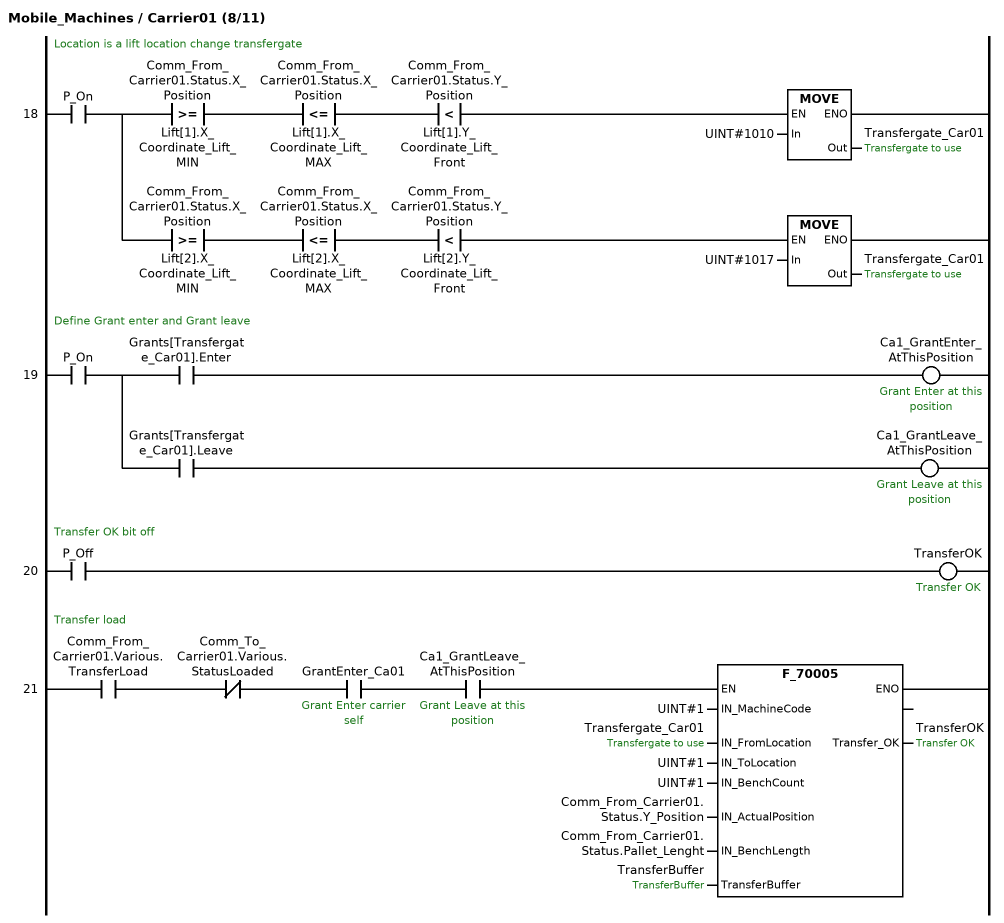
(* [picture p30: Mobile_Machines / Carrier01, rungs 18-21] *)
(* Rung 18: Location is a lift location change transfergate *)
IF P_On AND (Comm_From_Carrier01.Status.X_Position >= Lift[1].X_Coordinate_Lift_MIN) AND (Comm_From_Carrier01.Status.X_Position <= Lift[1].X_Coordinate_Lift_MAX) AND (Comm_From_Carrier01.Status.Y_Position < Lift[1].Y_Coordinate_Lift_Front) THEN
    Transfergate_Car01 := UINT#1010;
END_IF;
IF P_On AND (Comm_From_Carrier01.Status.X_Position >= Lift[2].X_Coordinate_Lift_MIN) AND (Comm_From_Carrier01.Status.X_Position <= Lift[2].X_Coordinate_Lift_MAX) AND (Comm_From_Carrier01.Status.Y_Position < Lift[2].Y_Coordinate_Lift_Front) THEN
    Transfergate_Car01 := UINT#1017;
END_IF;
(* Rung 19: Define Grant enter and Grant leave *)
Ca1_GrantEnter_AtThisPosition := P_On AND Grants[Transfergate_Car01].Enter;
Ca1_GrantLeave_AtThisPosition := P_On AND Grants[Transfergate_Car01].Leave;
(* Rung 20: Transfer OK bit off *)
TransferOK := P_Off;
(* Rung 21: Transfer load *)
IF Comm_From_Carrier01.Various.TransferLoad AND NOT Comm_To_Carrier01.Various.StatusLoaded AND GrantEnter_Ca01 AND Ca1_GrantLeave_AtThisPosition THEN
    F_70005(IN_MachineCode := UINT#1, IN_FromLocation := Transfergate_Car01, IN_ToLocation := UINT#1, IN_BenchCount := UINT#1, IN_ActualPosition := Comm_From_Carrier01.Status.Y_Position, IN_BenchLength := Comm_From_Carrier01.Status.Pallet_Lenght, TransferBuffer := TransferBuffer, Transfer_OK => TransferOK);
END_IF;

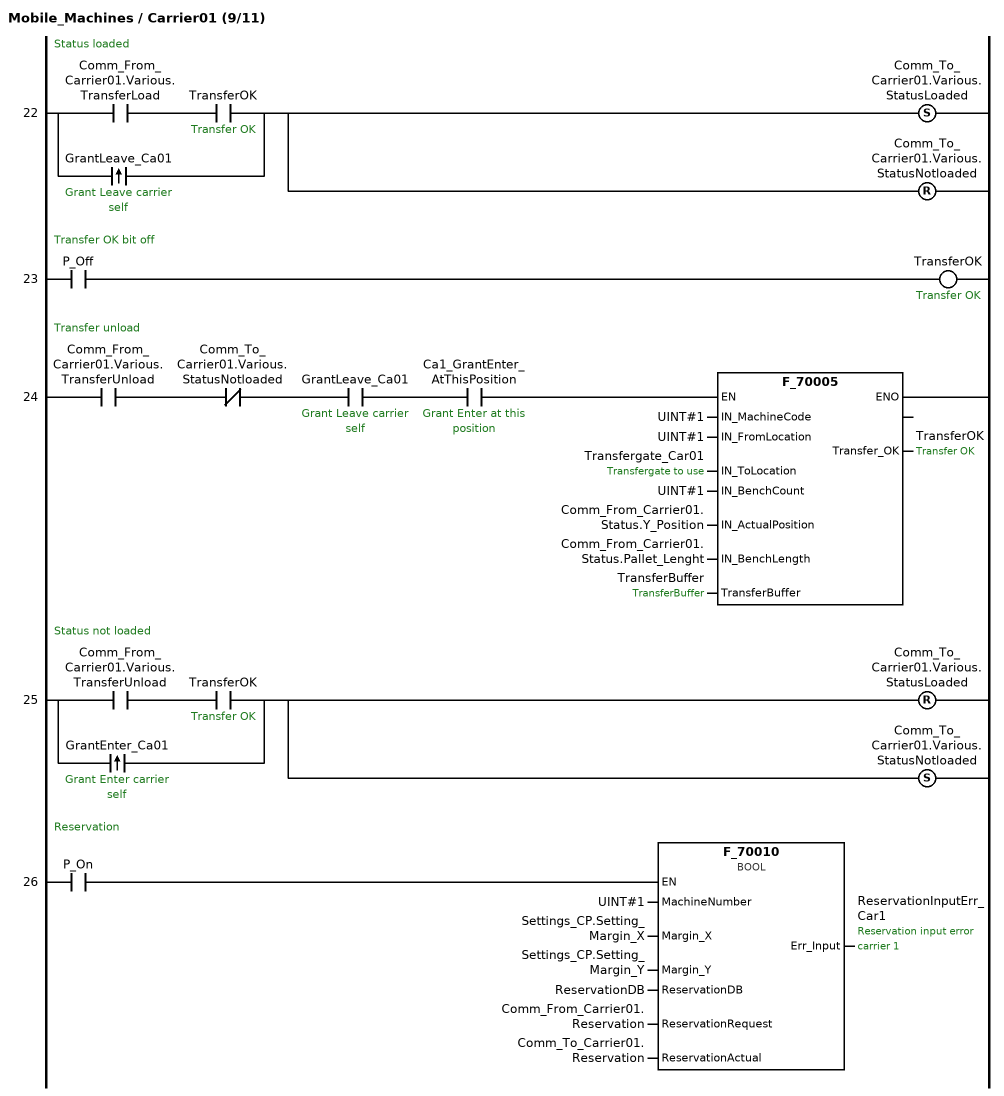
(* Rung 22: Status loaded *)
_e5(CLK := GrantLeave_Ca01);
_p6 := (Comm_From_Carrier01.Various.TransferLoad AND TransferOK) OR _e5.Q;
IF _p6 THEN
    Comm_To_Carrier01.Various.StatusLoaded := TRUE;
    Comm_To_Carrier01.Various.StatusNotloaded := FALSE;
END_IF;
(* Rung 23: Transfer OK bit off *)
TransferOK := P_Off;
(* Rung 24: Transfer unload *)
IF Comm_From_Carrier01.Various.TransferUnload AND NOT Comm_To_Carrier01.Various.StatusNotloaded AND GrantLeave_Ca01 AND Ca1_GrantEnter_AtThisPosition THEN
    F_70005(IN_MachineCode := UINT#1, IN_FromLocation := UINT#1, IN_ToLocation := Transfergate_Car01, IN_BenchCount := UINT#1, IN_ActualPosition := Comm_From_Carrier01.Status.Y_Position, IN_BenchLength := Comm_From_Carrier01.Status.Pallet_Lenght, TransferBuffer := TransferBuffer, Transfer_OK => TransferOK);
END_IF;
(* Rung 25: Status not loaded *)
_e7(CLK := GrantEnter_Ca01);
_p8 := (Comm_From_Carrier01.Various.TransferUnload AND TransferOK) OR _e7.Q;
IF _p8 THEN
    Comm_To_Carrier01.Various.StatusLoaded := FALSE;
    Comm_To_Carrier01.Various.StatusNotloaded := TRUE;
END_IF;
(* Rung 26: Reservation *)
_t9 := FALSE;
IF P_On THEN _t9 := F_70010(MachineNumber := UINT#1, Margin_X := Settings_CP.Setting_Margin_X, Margin_Y := Settings_CP.Setting_Margin_Y, ReservationDB := ReservationDB, ReservationRequest := Comm_From_Carrier01.Reservation, ReservationActual := Comm_To_Carrier01.Reservation, Err_Input => ReservationInputErr_Car1); END_IF;

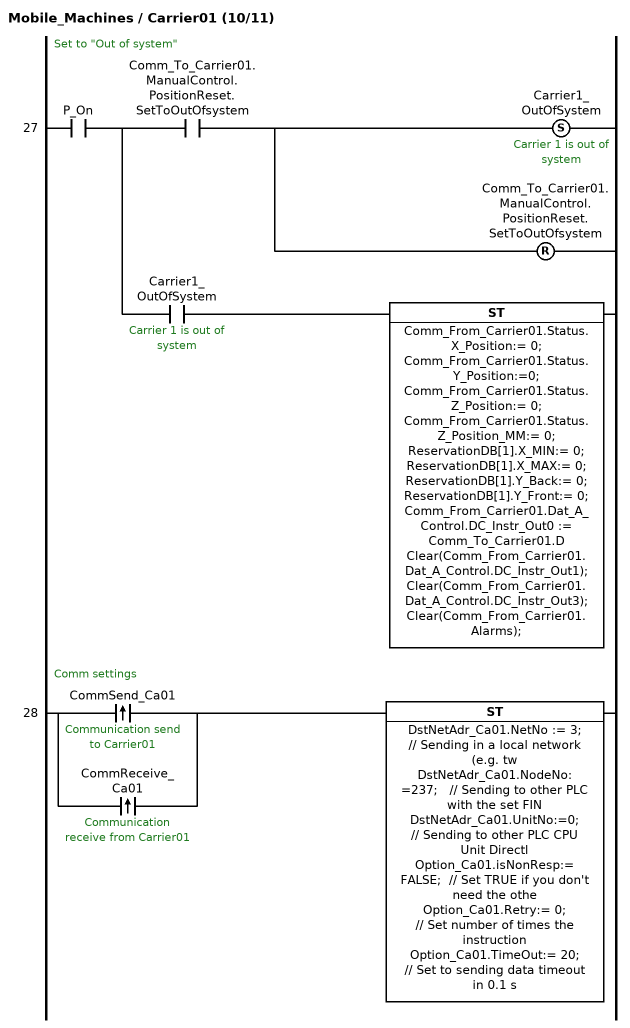
(* Rung 27: Set to "Out of system" *)
_p10 := P_On AND Comm_To_Carrier01.ManualControl.PositionReset.SetToOutOfsystem;
IF _p10 THEN
    Carrier1_OutOfSystem := TRUE;
    Comm_To_Carrier01.ManualControl.PositionReset.SetToOutOfsystem := FALSE;
END_IF;
IF P_On AND Carrier1_OutOfSystem THEN
    Comm_From_Carrier01.Status.X_Position:= 0;
    Comm_From_Carrier01.Status.Y_Position:=0;
    Comm_From_Carrier01.Status.Z_Position:= 0;
    Comm_From_Carrier01.Status.Z_Position_MM:= 0;
    
    ReservationDB[1].X_MIN:= 0;
    ReservationDB[1].X_MAX:= 0;
    ReservationDB[1].Y_Back:= 0;
    ReservationDB[1].Y_Front:= 0;
    
    Comm_From_Carrier01.Dat_A_Control.DC_Instr_Out0 := Comm_To_Carrier01.Dat_A_Control.Instr_Sequencenumber;
    Clear(Comm_From_Carrier01.Dat_A_Control.DC_Instr_Out1);
    Clear(Comm_From_Carrier01.Dat_A_Control.DC_Instr_Out3);
    Clear(Comm_From_Carrier01.Alarms);
END_IF;
(* Rung 28: Comm settings *)
_e11(CLK := CommSend_Ca01);
_e12(CLK := CommReceive_Ca01);
IF _e11.Q OR _e12.Q THEN
    DstNetAdr_Ca01.NetNo := 3;			// Sending in a local network (e.g. two PLCs connected by Ethernet LAN vai a hub)
    DstNetAdr_Ca01.NodeNo:=237;		// Sending to other PLC with the set FINS Node NUmber (depending on the other PLC)
    DstNetAdr_Ca01.UnitNo:=0;			// Sending to other PLC CPU Unit Directly
    
    Option_Ca01.isNonResp:= FALSE; 	// Set TRUE if you don't need the other CPU to reply back, otherwise set to FALSE
    Option_Ca01.Retry:= 0;					// Set number of times the instruction will retry sending if it failed to send data
    Option_Ca01.TimeOut:= 20;			// Set to sending data timeout in 0.1 s unit (e.g. 20 = 2 secs)
END_IF;

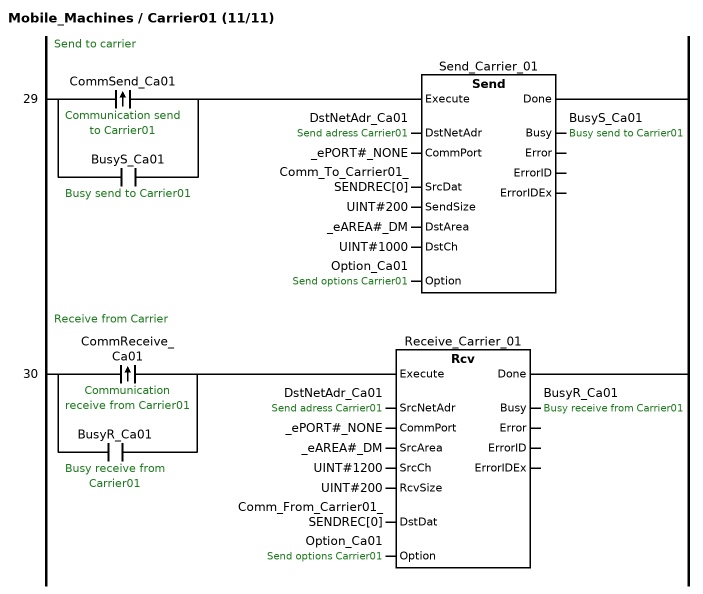
(* Rung 29: Send to carrier *)
_e13(CLK := CommSend_Ca01);
Send_Carrier_01(Execute := _e13.Q OR BusyS_Ca01, DstNetAdr := DstNetAdr_Ca01, CommPort := _ePORT#_NONE, SrcDat := Comm_To_Carrier01_SENDREC[0], SendSize := UINT#200, DstArea := _eAREA#_DM, DstCh := UINT#1000, Option := Option_Ca01, Busy => BusyS_Ca01);
(* Rung 30: Receive from Carrier *)
_e14(CLK := CommReceive_Ca01);
Receive_Carrier_01(Execute := _e14.Q OR BusyR_Ca01, SrcNetAdr := DstNetAdr_Ca01, CommPort := _ePORT#_NONE, SrcArea := _eAREA#_DM, SrcCh := UINT#1200, RcvSize := UINT#200, DstDat := Comm_From_Carrier01_SENDREC[0], Option := Option_Ca01, Busy => BusyR_Ca01);

(* Section Carrier02: ladder, written here as Structured Text *)

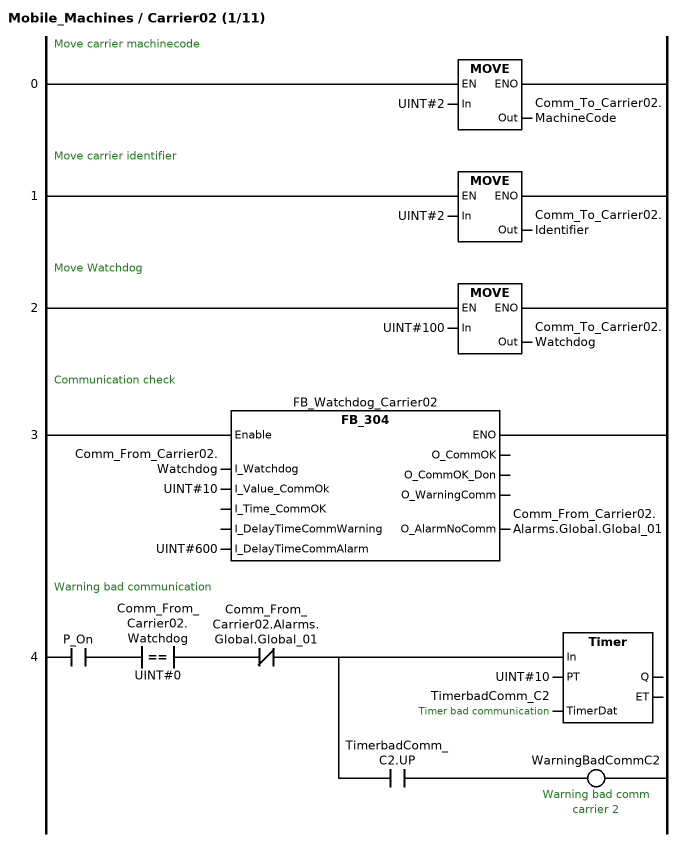
(* Rung 0: Move carrier machinecode *)
Comm_To_Carrier02.MachineCode := UINT#2;
(* Rung 1: Move carrier identifier *)
Comm_To_Carrier02.Identifier := UINT#2;
(* Rung 2: Move Watchdog *)
Comm_To_Carrier02.Watchdog := UINT#100;
(* Rung 3: Communication check *)
FB_Watchdog_Carrier02(Enable := TRUE, I_Watchdog := Comm_From_Carrier02.Watchdog, I_Value_CommOk := UINT#10, I_DelayTimeCommAlarm := UINT#600, O_AlarmNoComm => Comm_From_Carrier02.Alarms.Global.Global_01);
(* Rung 4: Warning bad communication *)
_p15 := P_On AND (Comm_From_Carrier02.Watchdog = UINT#0) AND NOT Comm_From_Carrier02.Alarms.Global.Global_01;
_t16 := Timer(In := _p15, PT := UINT#10, TimerDat := TimerbadComm_C2);
WarningBadCommC2 := _p15 AND TimerbadComm_C2.UP;

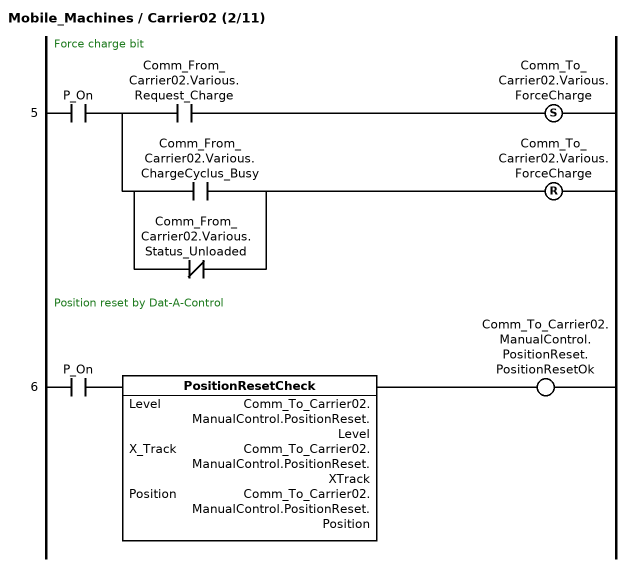
(* Rung 5: Force charge bit *)
IF P_On AND Comm_From_Carrier02.Various.Request_Charge THEN
    Comm_To_Carrier02.Various.ForceCharge := TRUE;
END_IF;
IF P_On AND (Comm_From_Carrier02.Various.ChargeCyclus_Busy OR NOT Comm_From_Carrier02.Various.Status_Unloaded) THEN
    Comm_To_Carrier02.Various.ForceCharge := FALSE;
END_IF;
(* Rung 6: Position reset by Dat-A-Control *)
Comm_To_Carrier02.ManualControl.PositionReset.PositionResetOk := P_On AND PositionResetCheck(Level := Comm_To_Carrier02.ManualControl.PositionReset.Level, X_Track := Comm_To_Carrier02.ManualControl.PositionReset.XTrack, Position := Comm_To_Carrier02.ManualControl.PositionReset.Position);

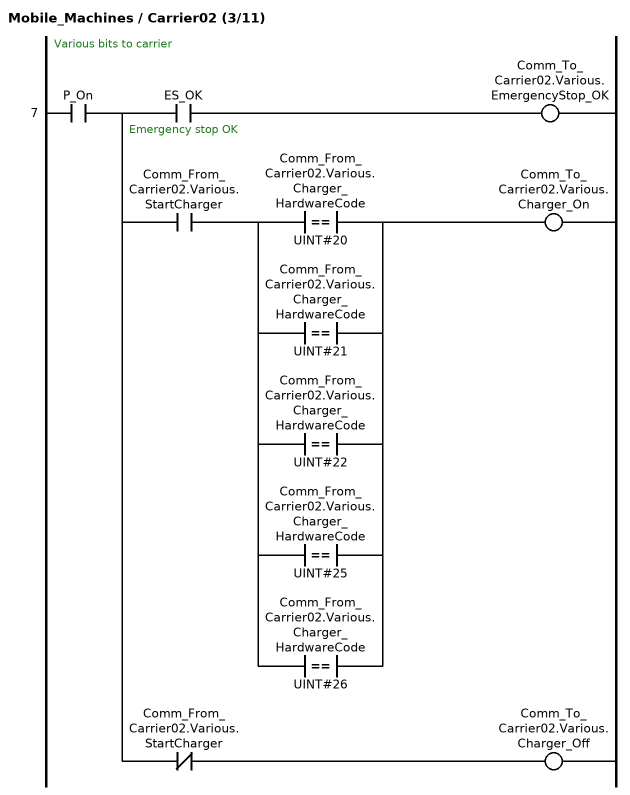
(* Rung 7: Various bits to carrier *)
Comm_To_Carrier02.Various.EmergencyStop_OK := P_On AND ES_OK;
Comm_To_Carrier02.Various.Charger_On := P_On AND Comm_From_Carrier02.Various.StartCharger AND ((Comm_From_Carrier02.Various.Charger_HardwareCode = UINT#20) OR (Comm_From_Carrier02.Various.Charger_HardwareCode = UINT#21) OR (Comm_From_Carrier02.Various.Charger_HardwareCode = UINT#22) OR (Comm_From_Carrier02.Various.Charger_HardwareCode = UINT#25) OR (Comm_From_Carrier02.Various.Charger_HardwareCode = UINT#26));
Comm_To_Carrier02.Various.Charger_Off := P_On AND NOT Comm_From_Carrier02.Various.StartCharger;

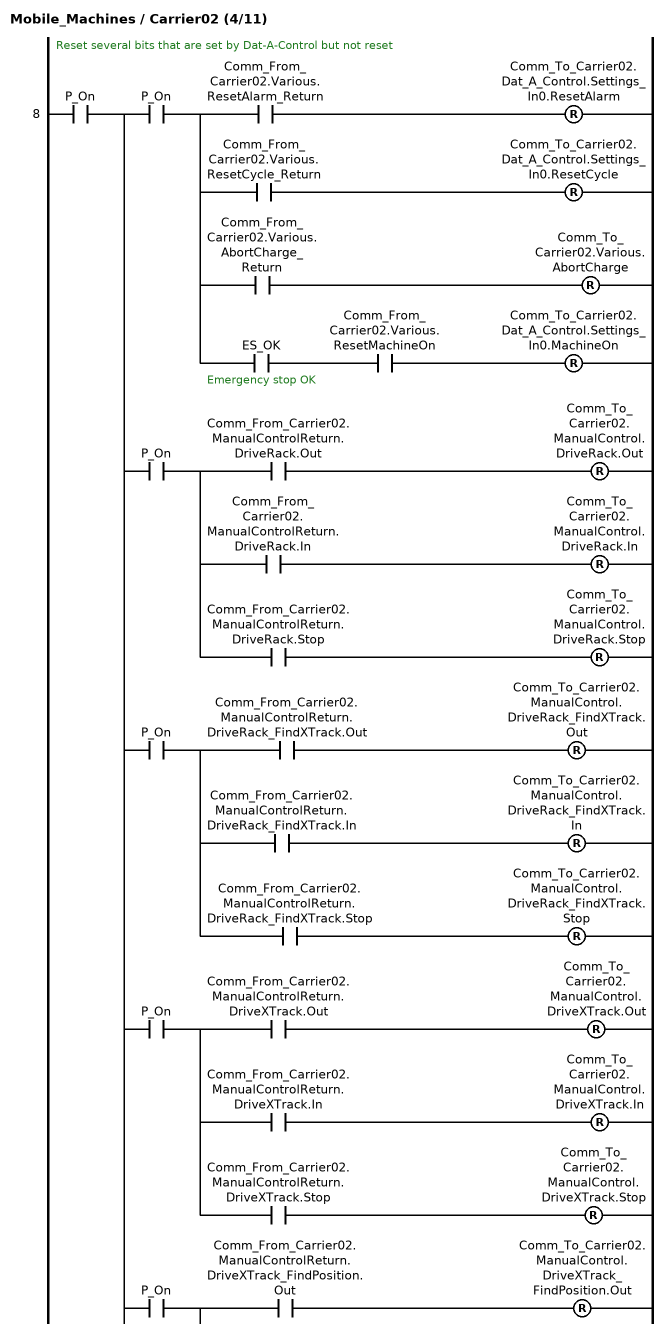

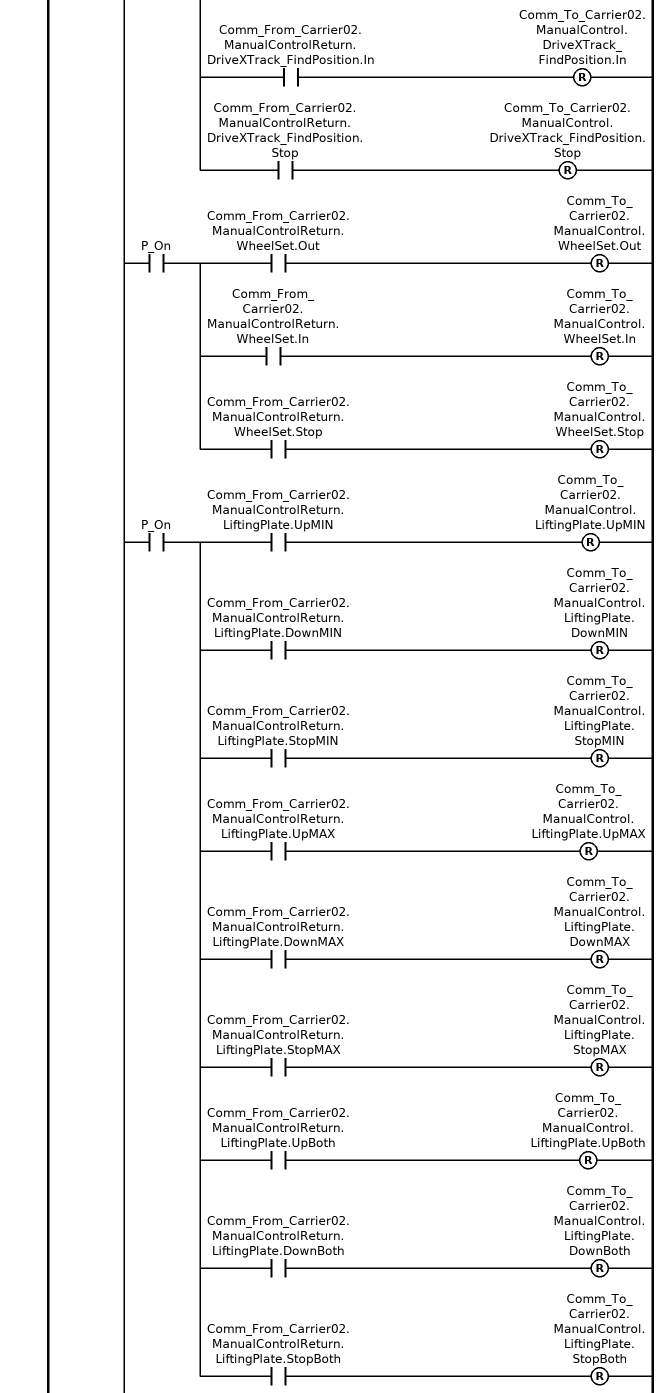

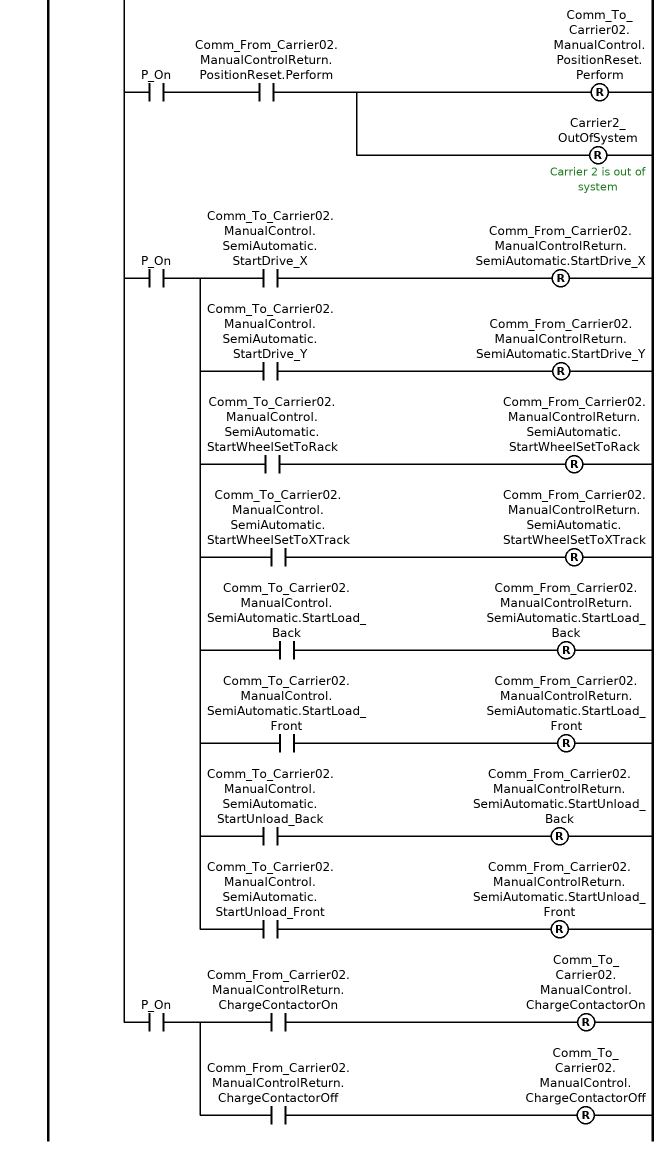
(* Rung 8: Reset several bits that are set by Dat-A-Control but not reset *)
IF P_On AND P_On AND Comm_From_Carrier02.Various.ResetAlarm_Return THEN
    Comm_To_Carrier02.Dat_A_Control.Settings_In0.ResetAlarm := FALSE;
END_IF;
IF P_On AND P_On AND Comm_From_Carrier02.Various.ResetCycle_Return THEN
    Comm_To_Carrier02.Dat_A_Control.Settings_In0.ResetCycle := FALSE;
END_IF;
IF P_On AND P_On AND Comm_From_Carrier02.Various.AbortCharge_Return THEN
    Comm_To_Carrier02.Various.AbortCharge := FALSE;
END_IF;
IF P_On AND P_On AND ES_OK AND Comm_From_Carrier02.Various.ResetMachineOn THEN
    Comm_To_Carrier02.Dat_A_Control.Settings_In0.MachineOn := FALSE;
END_IF;
IF P_On AND P_On AND Comm_From_Carrier02.ManualControlReturn.DriveRack.Out THEN
    Comm_To_Carrier02.ManualControl.DriveRack.Out := FALSE;
END_IF;
IF P_On AND P_On AND Comm_From_Carrier02.ManualControlReturn.DriveRack.In THEN
    Comm_To_Carrier02.ManualControl.DriveRack.In := FALSE;
END_IF;
IF P_On AND P_On AND Comm_From_Carrier02.ManualControlReturn.DriveRack.Stop THEN
    Comm_To_Carrier02.ManualControl.DriveRack.Stop := FALSE;
END_IF;
IF P_On AND P_On AND Comm_From_Carrier02.ManualControlReturn.DriveRack_FindXTrack.Out THEN
    Comm_To_Carrier02.ManualControl.DriveRack_FindXTrack.Out := FALSE;
END_IF;
IF P_On AND P_On AND Comm_From_Carrier02.ManualControlReturn.DriveRack_FindXTrack.In THEN
    Comm_To_Carrier02.ManualControl.DriveRack_FindXTrack.In := FALSE;
END_IF;
IF P_On AND P_On AND Comm_From_Carrier02.ManualControlReturn.DriveRack_FindXTrack.Stop THEN
    Comm_To_Carrier02.ManualControl.DriveRack_FindXTrack.Stop := FALSE;
END_IF;
IF P_On AND P_On AND Comm_From_Carrier02.ManualControlReturn.DriveXTrack.Out THEN
    Comm_To_Carrier02.ManualControl.DriveXTrack.Out := FALSE;
END_IF;
IF P_On AND P_On AND Comm_From_Carrier02.ManualControlReturn.DriveXTrack.In THEN
    Comm_To_Carrier02.ManualControl.DriveXTrack.In := FALSE;
END_IF;
IF P_On AND P_On AND Comm_From_Carrier02.ManualControlReturn.DriveXTrack.Stop THEN
    Comm_To_Carrier02.ManualControl.DriveXTrack.Stop := FALSE;
END_IF;
IF P_On AND P_On AND Comm_From_Carrier02.ManualControlReturn.DriveXTrack_FindPosition.Out THEN
    Comm_To_Carrier02.ManualControl.DriveXTrack_FindPosition.Out := FALSE;
END_IF;
IF P_On AND P_On AND Comm_From_Carrier02.ManualControlReturn.DriveXTrack_FindPosition.In THEN
    Comm_To_Carrier02.ManualControl.DriveXTrack_FindPosition.In := FALSE;
END_IF;
IF P_On AND P_On AND Comm_From_Carrier02.ManualControlReturn.DriveXTrack_FindPosition.Stop THEN
    Comm_To_Carrier02.ManualControl.DriveXTrack_FindPosition.Stop := FALSE;
END_IF;
IF P_On AND P_On AND Comm_From_Carrier02.ManualControlReturn.WheelSet.Out THEN
    Comm_To_Carrier02.ManualControl.WheelSet.Out := FALSE;
END_IF;
IF P_On AND P_On AND Comm_From_Carrier02.ManualControlReturn.WheelSet.In THEN
    Comm_To_Carrier02.ManualControl.WheelSet.In := FALSE;
END_IF;
IF P_On AND P_On AND Comm_From_Carrier02.ManualControlReturn.WheelSet.Stop THEN
    Comm_To_Carrier02.ManualControl.WheelSet.Stop := FALSE;
END_IF;
IF P_On AND P_On AND Comm_From_Carrier02.ManualControlReturn.LiftingPlate.UpMIN THEN
    Comm_To_Carrier02.ManualControl.LiftingPlate.UpMIN := FALSE;
END_IF;
IF P_On AND P_On AND Comm_From_Carrier02.ManualControlReturn.LiftingPlate.DownMIN THEN
    Comm_To_Carrier02.ManualControl.LiftingPlate.DownMIN := FALSE;
END_IF;
IF P_On AND P_On AND Comm_From_Carrier02.ManualControlReturn.LiftingPlate.StopMIN THEN
    Comm_To_Carrier02.ManualControl.LiftingPlate.StopMIN := FALSE;
END_IF;
IF P_On AND P_On AND Comm_From_Carrier02.ManualControlReturn.LiftingPlate.UpMAX THEN
    Comm_To_Carrier02.ManualControl.LiftingPlate.UpMAX := FALSE;
END_IF;
IF P_On AND P_On AND Comm_From_Carrier02.ManualControlReturn.LiftingPlate.DownMAX THEN
    Comm_To_Carrier02.ManualControl.LiftingPlate.DownMAX := FALSE;
END_IF;
IF P_On AND P_On AND Comm_From_Carrier02.ManualControlReturn.LiftingPlate.StopMAX THEN
    Comm_To_Carrier02.ManualControl.LiftingPlate.StopMAX := FALSE;
END_IF;
IF P_On AND P_On AND Comm_From_Carrier02.ManualControlReturn.LiftingPlate.UpBoth THEN
    Comm_To_Carrier02.ManualControl.LiftingPlate.UpBoth := FALSE;
END_IF;
IF P_On AND P_On AND Comm_From_Carrier02.ManualControlReturn.LiftingPlate.DownBoth THEN
    Comm_To_Carrier02.ManualControl.LiftingPlate.DownBoth := FALSE;
END_IF;
IF P_On AND P_On AND Comm_From_Carrier02.ManualControlReturn.LiftingPlate.StopBoth THEN
    Comm_To_Carrier02.ManualControl.LiftingPlate.StopBoth := FALSE;
END_IF;
_p17 := P_On AND P_On AND Comm_From_Carrier02.ManualControlReturn.PositionReset.Perform;
IF _p17 THEN
    Comm_To_Carrier02.ManualControl.PositionReset.Perform := FALSE;
    Carrier2_OutOfSystem := FALSE;
END_IF;
IF P_On AND P_On AND Comm_To_Carrier02.ManualControl.SemiAutomatic.StartDrive_X THEN
    Comm_From_Carrier02.ManualControlReturn.SemiAutomatic.StartDrive_X := FALSE;
END_IF;
IF P_On AND P_On AND Comm_To_Carrier02.ManualControl.SemiAutomatic.StartDrive_Y THEN
    Comm_From_Carrier02.ManualControlReturn.SemiAutomatic.StartDrive_Y := FALSE;
END_IF;
IF P_On AND P_On AND Comm_To_Carrier02.ManualControl.SemiAutomatic.StartWheelSetToRack THEN
    Comm_From_Carrier02.ManualControlReturn.SemiAutomatic.StartWheelSetToRack := FALSE;
END_IF;
IF P_On AND P_On AND Comm_To_Carrier02.ManualControl.SemiAutomatic.StartWheelSetToXTrack THEN
    Comm_From_Carrier02.ManualControlReturn.SemiAutomatic.StartWheelSetToXTrack := FALSE;
END_IF;
IF P_On AND P_On AND Comm_To_Carrier02.ManualControl.SemiAutomatic.StartLoad_Back THEN
    Comm_From_Carrier02.ManualControlReturn.SemiAutomatic.StartLoad_Back := FALSE;
END_IF;
IF P_On AND P_On AND Comm_To_Carrier02.ManualControl.SemiAutomatic.StartLoad_Front THEN
    Comm_From_Carrier02.ManualControlReturn.SemiAutomatic.StartLoad_Front := FALSE;
END_IF;
IF P_On AND P_On AND Comm_To_Carrier02.ManualControl.SemiAutomatic.StartUnload_Back THEN
    Comm_From_Carrier02.ManualControlReturn.SemiAutomatic.StartUnload_Back := FALSE;
END_IF;
IF P_On AND P_On AND Comm_To_Carrier02.ManualControl.SemiAutomatic.StartUnload_Front THEN
    Comm_From_Carrier02.ManualControlReturn.SemiAutomatic.StartUnload_Front := FALSE;
END_IF;
IF P_On AND P_On AND Comm_From_Carrier02.ManualControlReturn.ChargeContactorOn THEN
    Comm_To_Carrier02.ManualControl.ChargeContactorOn := FALSE;
END_IF;
IF P_On AND P_On AND Comm_From_Carrier02.ManualControlReturn.ChargeContactorOff THEN
    Comm_To_Carrier02.ManualControl.ChargeContactorOff := FALSE;
END_IF;

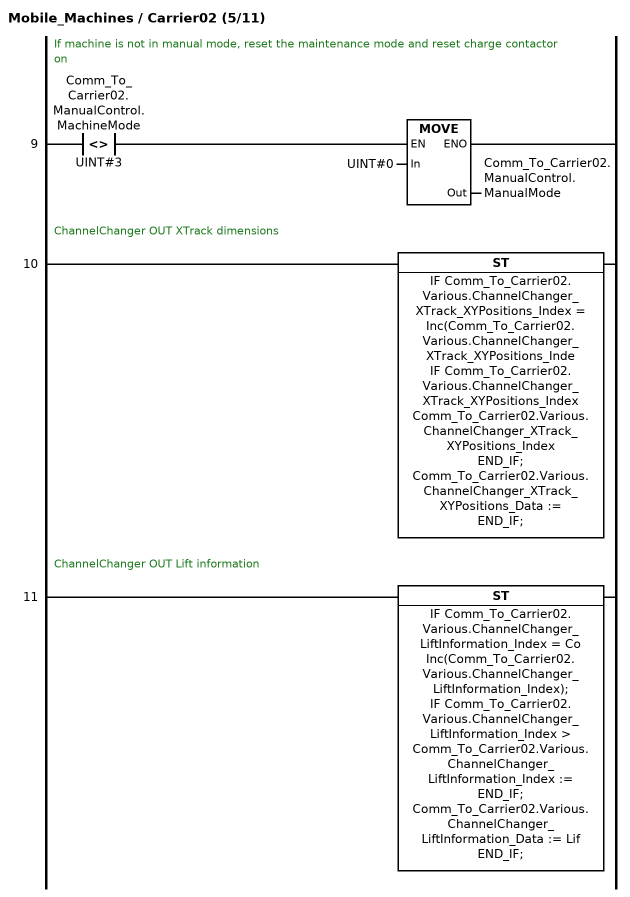
(* Rung 9: If machine is not in manual mode, reset the maintenance mode and reset charge contactor on *)
IF Comm_To_Carrier02.ManualControl.MachineMode <> UINT#3 THEN
    Comm_To_Carrier02.ManualControl.ManualMode := UINT#0;
END_IF;
(* Rung 10: ChannelChanger OUT XTrack dimensions *)
IF Comm_To_Carrier02.Various.ChannelChanger_XTrack_XYPositions_Index = Comm_From_Carrier02.Various.ChannelChanger_XTrack_XYPositions_Index THEN
	Inc(Comm_To_Carrier02.Various.ChannelChanger_XTrack_XYPositions_Index);
	IF Comm_To_Carrier02.Various.ChannelChanger_XTrack_XYPositions_Index > 199 THEN
		Comm_To_Carrier02.Various.ChannelChanger_XTrack_XYPositions_Index := 0;
	END_IF;
	Comm_To_Carrier02.Various.ChannelChanger_XTrack_XYPositions_Data := XTrack_XYPositions_Array[Comm_To_Carrier02.Various.ChannelChanger_XTrack_XYPositions_Index];
END_IF;
(* Rung 11: ChannelChanger OUT Lift information *)
IF Comm_To_Carrier02.Various.ChannelChanger_LiftInformation_Index = Comm_From_Carrier02.Various.ChannelChanger_LiftInformation_Index THEN
	Inc(Comm_To_Carrier02.Various.ChannelChanger_LiftInformation_Index);
	IF Comm_To_Carrier02.Various.ChannelChanger_LiftInformation_Index > 99 THEN
		Comm_To_Carrier02.Various.ChannelChanger_LiftInformation_Index := 0;
	END_IF;
	Comm_To_Carrier02.Various.ChannelChanger_LiftInformation_Data := Lift_Array[Comm_To_Carrier02.Various.ChannelChanger_LiftInformation_Index];
END_IF;

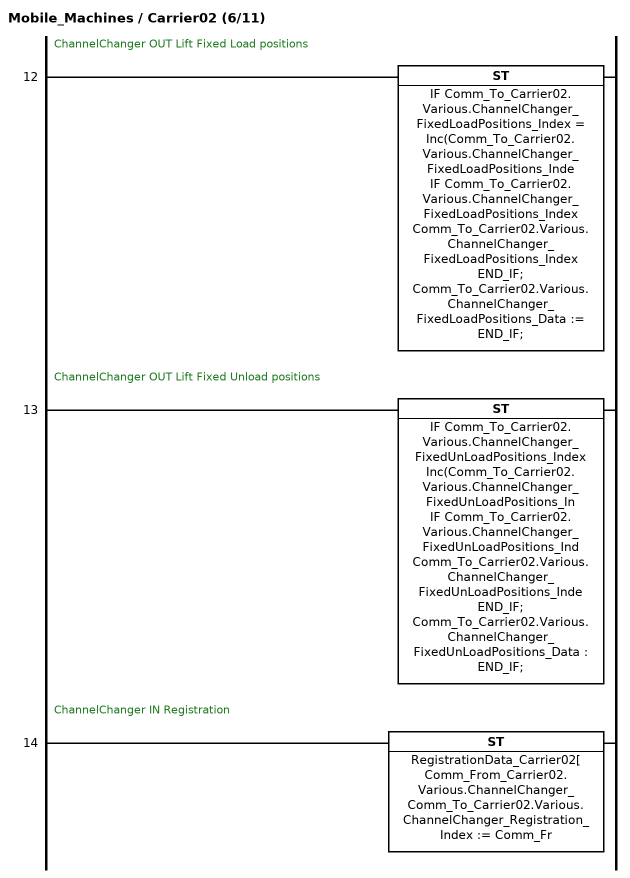
(* Rung 12: ChannelChanger OUT Lift Fixed Load positions *)
IF Comm_To_Carrier02.Various.ChannelChanger_FixedLoadPositions_Index = Comm_From_Carrier02.Various.ChannelChanger_FixedLoadPositions_Index THEN
	Inc(Comm_To_Carrier02.Various.ChannelChanger_FixedLoadPositions_Index);
	IF Comm_To_Carrier02.Various.ChannelChanger_FixedLoadPositions_Index > 199 THEN
		Comm_To_Carrier02.Various.ChannelChanger_FixedLoadPositions_Index := 0;
	END_IF;
	Comm_To_Carrier02.Various.ChannelChanger_FixedLoadPositions_Data := FixedLoadPosition_Array[Comm_To_Carrier02.Various.ChannelChanger_FixedLoadPositions_Index];
END_IF;
(* Rung 13: ChannelChanger OUT Lift Fixed Unload positions *)
IF Comm_To_Carrier02.Various.ChannelChanger_FixedUnLoadPositions_Index = Comm_From_Carrier02.Various.ChannelChanger_FixedUnLoadPositions_Index THEN
	Inc(Comm_To_Carrier02.Various.ChannelChanger_FixedUnLoadPositions_Index);
	IF Comm_To_Carrier02.Various.ChannelChanger_FixedUnLoadPositions_Index > 199 THEN
		Comm_To_Carrier02.Various.ChannelChanger_FixedUnLoadPositions_Index := 0;
	END_IF;
	Comm_To_Carrier02.Various.ChannelChanger_FixedUnLoadPositions_Data := FixedUnloadPosition_Array[Comm_To_Carrier02.Various.ChannelChanger_FixedUnLoadPositions_Index];
END_IF;
(* Rung 14: ChannelChanger IN Registration *)
RegistrationData_Carrier02[Comm_From_Carrier02.Various.ChannelChanger_Registration_Index] := Comm_From_Carrier02.Various.ChannelChanger_Registration_Data;
Comm_To_Carrier02.Various.ChannelChanger_Registration_Index := Comm_From_Carrier02.Various.ChannelChanger_Registration_Index;

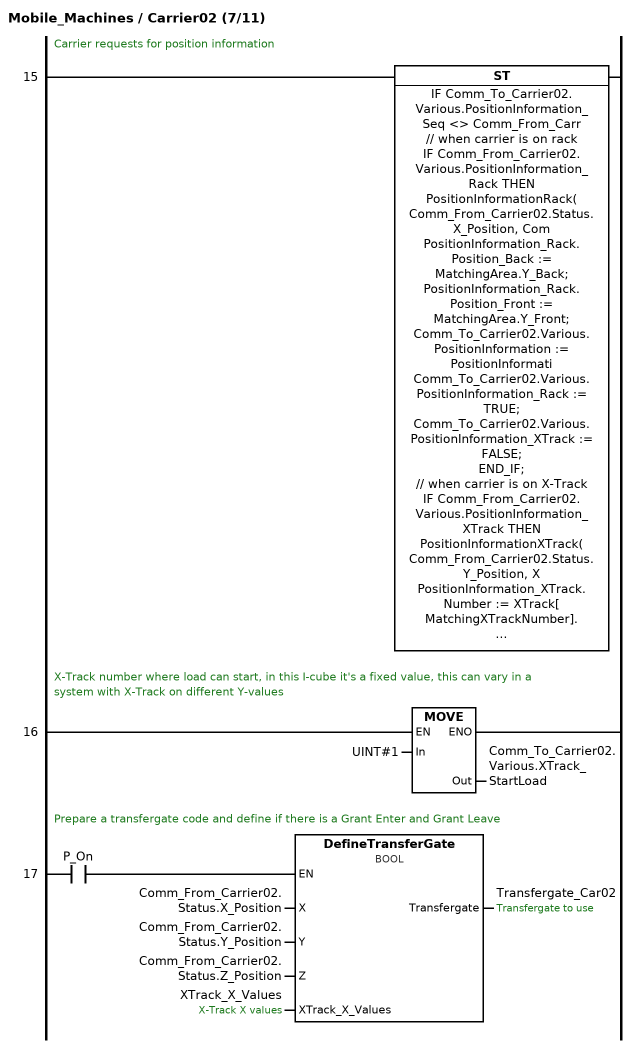
(* Rung 15: Carrier requests for position information *)
IF Comm_To_Carrier02.Various.PositionInformation_Seq <> Comm_From_Carrier02.Various.PositionInformation_Seq THEN
	// when carrier is on rack
	IF Comm_From_Carrier02.Various.PositionInformation_Rack THEN
		PositionInformationRack(Comm_From_Carrier02.Status.X_Position, Comm_From_Carrier02.Status.Y_Position, Comm_From_Carrier02.Status.Z_Position, Settings_CP.Margin_AreaCompare, Area, MatchingArea);
		PositionInformation_Rack.Position_Back := MatchingArea.Y_Back;
		PositionInformation_Rack.Position_Front := MatchingArea.Y_Front;
		Comm_To_Carrier02.Various.PositionInformation := PositionInformation_Rough;
		Comm_To_Carrier02.Various.PositionInformation_Rack := TRUE;
		Comm_To_Carrier02.Various.PositionInformation_XTrack := FALSE;
	END_IF;
	
	// when carrier is on X-Track
	IF Comm_From_Carrier02.Various.PositionInformation_XTrack THEN
		PositionInformationXTrack(Comm_From_Carrier02.Status.Y_Position, XTrack_Y_Values, MatchingXTrackNumber);
		PositionInformation_XTrack.Number := XTrack[MatchingXTrackNumber].XTrack_Number;
		PositionInformation_XTrack.Position_MIN := XTrack[MatchingXTrackNumber].MinimumPosition;
		PositionInformation_XTrack.Position_MAX := XTrack[MatchingXTrackNumber].MaximumPosition;
		Comm_To_Carrier02.Various.PositionInformation := PositionInformation_Rough;
		Comm_To_Carrier02.Various.PositionInformation_Rack := FALSE;
		Comm_To_Carrier02.Various.PositionInformation_XTrack := TRUE;
	END_IF;
	
	Comm_To_Carrier02.Various.PositionInformation_Seq := Comm_From_Carrier02.Various.PositionInformation_Seq;
	
END_IF;
(* Rung 16: X-Track number where load can start, in this I-cube it's a fixed value, this can vary in a system with X-Track on different Y-values *)
Comm_To_Carrier02.Various.XTrack_StartLoad := UINT#1;
(* Rung 17: Prepare a transfergate code and define if there is a Grant Enter and Grant Leave *)
_t18 := FALSE;
IF P_On THEN _t18 := DefineTransferGate(X := Comm_From_Carrier02.Status.X_Position, Y := Comm_From_Carrier02.Status.Y_Position, Z := Comm_From_Carrier02.Status.Z_Position, XTrack_X_Values := XTrack_X_Values, Transfergate => Transfergate_Car02); END_IF;

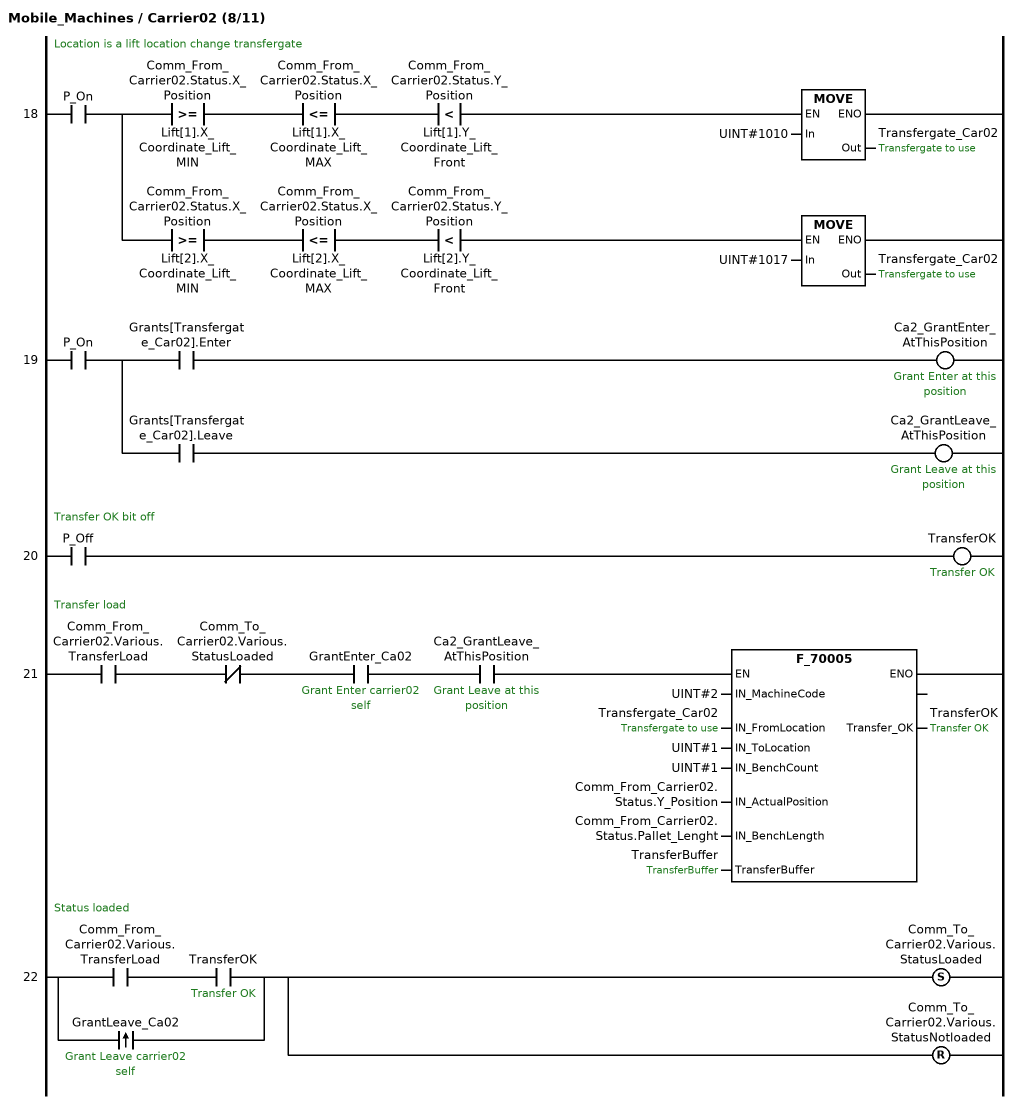
(* Rung 18: Location is a lift location change transfergate *)
IF P_On AND (Comm_From_Carrier02.Status.X_Position >= Lift[1].X_Coordinate_Lift_MIN) AND (Comm_From_Carrier02.Status.X_Position <= Lift[1].X_Coordinate_Lift_MAX) AND (Comm_From_Carrier02.Status.Y_Position < Lift[1].Y_Coordinate_Lift_Front) THEN
    Transfergate_Car02 := UINT#1010;
END_IF;
IF P_On AND (Comm_From_Carrier02.Status.X_Position >= Lift[2].X_Coordinate_Lift_MIN) AND (Comm_From_Carrier02.Status.X_Position <= Lift[2].X_Coordinate_Lift_MAX) AND (Comm_From_Carrier02.Status.Y_Position < Lift[2].Y_Coordinate_Lift_Front) THEN
    Transfergate_Car02 := UINT#1017;
END_IF;
(* Rung 19 *)
Ca2_GrantEnter_AtThisPosition := P_On AND Grants[Transfergate_Car02].Enter;
Ca2_GrantLeave_AtThisPosition := P_On AND Grants[Transfergate_Car02].Leave;
(* Rung 20: Transfer OK bit off *)
TransferOK := P_Off;
(* Rung 21: Transfer load *)
IF Comm_From_Carrier02.Various.TransferLoad AND NOT Comm_To_Carrier02.Various.StatusLoaded AND GrantEnter_Ca02 AND Ca2_GrantLeave_AtThisPosition THEN
    F_70005(IN_MachineCode := UINT#2, IN_FromLocation := Transfergate_Car02, IN_ToLocation := UINT#1, IN_BenchCount := UINT#1, IN_ActualPosition := Comm_From_Carrier02.Status.Y_Position, IN_BenchLength := Comm_From_Carrier02.Status.Pallet_Lenght, TransferBuffer := TransferBuffer, Transfer_OK => TransferOK);
END_IF;
(* Rung 22: Status loaded *)
_e19(CLK := GrantLeave_Ca02);
_p20 := (Comm_From_Carrier02.Various.TransferLoad AND TransferOK) OR _e19.Q;
IF _p20 THEN
    Comm_To_Carrier02.Various.StatusLoaded := TRUE;
    Comm_To_Carrier02.Various.StatusNotloaded := FALSE;
END_IF;

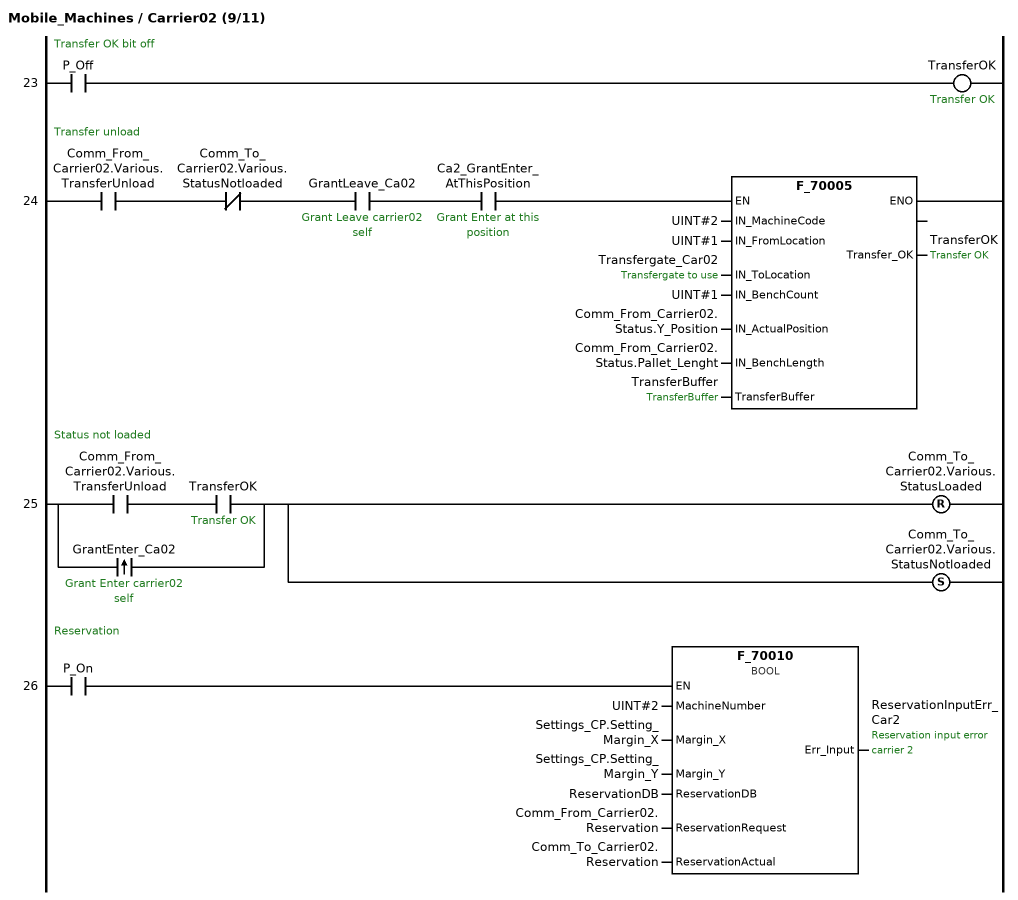
(* Rung 23: Transfer OK bit off *)
TransferOK := P_Off;
(* Rung 24: Transfer unload *)
IF Comm_From_Carrier02.Various.TransferUnload AND NOT Comm_To_Carrier02.Various.StatusNotloaded AND GrantLeave_Ca02 AND Ca2_GrantEnter_AtThisPosition THEN
    F_70005(IN_MachineCode := UINT#2, IN_FromLocation := UINT#1, IN_ToLocation := Transfergate_Car02, IN_BenchCount := UINT#1, IN_ActualPosition := Comm_From_Carrier02.Status.Y_Position, IN_BenchLength := Comm_From_Carrier02.Status.Pallet_Lenght, TransferBuffer := TransferBuffer, Transfer_OK => TransferOK);
END_IF;
(* Rung 25: Status not loaded *)
_e21(CLK := GrantEnter_Ca02);
_p22 := (Comm_From_Carrier02.Various.TransferUnload AND TransferOK) OR _e21.Q;
IF _p22 THEN
    Comm_To_Carrier02.Various.StatusLoaded := FALSE;
    Comm_To_Carrier02.Various.StatusNotloaded := TRUE;
END_IF;
(* Rung 26: Reservation *)
_t23 := FALSE;
IF P_On THEN _t23 := F_70010(MachineNumber := UINT#2, Margin_X := Settings_CP.Setting_Margin_X, Margin_Y := Settings_CP.Setting_Margin_Y, ReservationDB := ReservationDB, ReservationRequest := Comm_From_Carrier02.Reservation, ReservationActual := Comm_To_Carrier02.Reservation, Err_Input => ReservationInputErr_Car2); END_IF;

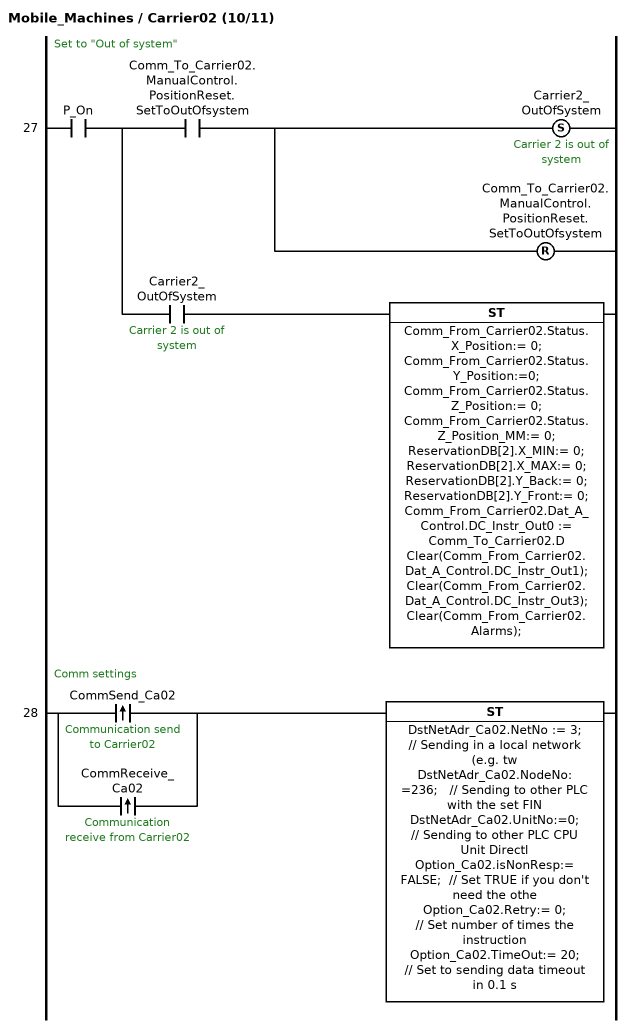
(* Rung 27: Set to "Out of system" *)
_p24 := P_On AND Comm_To_Carrier02.ManualControl.PositionReset.SetToOutOfsystem;
IF _p24 THEN
    Carrier2_OutOfSystem := TRUE;
    Comm_To_Carrier02.ManualControl.PositionReset.SetToOutOfsystem := FALSE;
END_IF;
IF P_On AND Carrier2_OutOfSystem THEN
    Comm_From_Carrier02.Status.X_Position:= 0;
    Comm_From_Carrier02.Status.Y_Position:=0;
    Comm_From_Carrier02.Status.Z_Position:= 0;
    Comm_From_Carrier02.Status.Z_Position_MM:= 0;
    
    ReservationDB[2].X_MIN:= 0;
    ReservationDB[2].X_MAX:= 0;
    ReservationDB[2].Y_Back:= 0;
    ReservationDB[2].Y_Front:= 0;
    
    Comm_From_Carrier02.Dat_A_Control.DC_Instr_Out0 := Comm_To_Carrier02.Dat_A_Control.Instr_Sequencenumber;
    Clear(Comm_From_Carrier02.Dat_A_Control.DC_Instr_Out1);
    Clear(Comm_From_Carrier02.Dat_A_Control.DC_Instr_Out3);
    Clear(Comm_From_Carrier02.Alarms);
END_IF;
(* Rung 28: Comm settings *)
_e25(CLK := CommSend_Ca02);
_e26(CLK := CommReceive_Ca02);
IF _e25.Q OR _e26.Q THEN
    DstNetAdr_Ca02.NetNo := 3;			// Sending in a local network (e.g. two PLCs connected by Ethernet LAN vai a hub)
    DstNetAdr_Ca02.NodeNo:=236;		// Sending to other PLC with the set FINS Node NUmber (depending on the other PLC)
    DstNetAdr_Ca02.UnitNo:=0;			// Sending to other PLC CPU Unit Directly
    
    Option_Ca02.isNonResp:= FALSE; 	// Set TRUE if you don't need the other CPU to reply back, otherwise set to FALSE
    Option_Ca02.Retry:= 0;					// Set number of times the instruction will retry sending if it failed to send data
    Option_Ca02.TimeOut:= 20;			// Set to sending data timeout in 0.1 s unit (e.g. 20 = 2 secs)
END_IF;

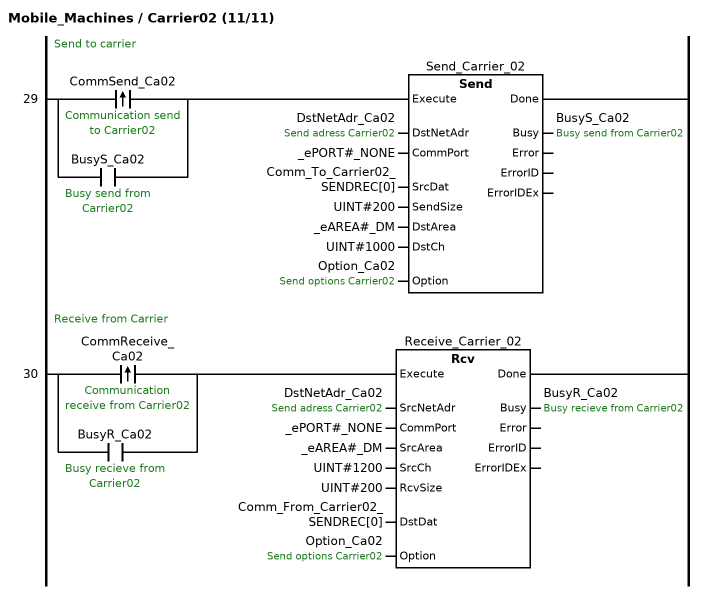
(* Rung 29: Send to carrier *)
_e27(CLK := CommSend_Ca02);
Send_Carrier_02(Execute := _e27.Q OR BusyS_Ca02, DstNetAdr := DstNetAdr_Ca02, CommPort := _ePORT#_NONE, SrcDat := Comm_To_Carrier02_SENDREC[0], SendSize := UINT#200, DstArea := _eAREA#_DM, DstCh := UINT#1000, Option := Option_Ca02, Busy => BusyS_Ca02);
(* Rung 30: Receive from Carrier *)
_e28(CLK := CommReceive_Ca02);
Receive_Carrier_02(Execute := _e28.Q OR BusyR_Ca02, SrcNetAdr := DstNetAdr_Ca02, CommPort := _ePORT#_NONE, SrcArea := _eAREA#_DM, SrcCh := UINT#1200, RcvSize := UINT#200, DstDat := Comm_From_Carrier02_SENDREC[0], Option := Option_Ca02, Busy => BusyR_Ca02);

(* Section Carrier03: ladder, written here as Structured Text *)

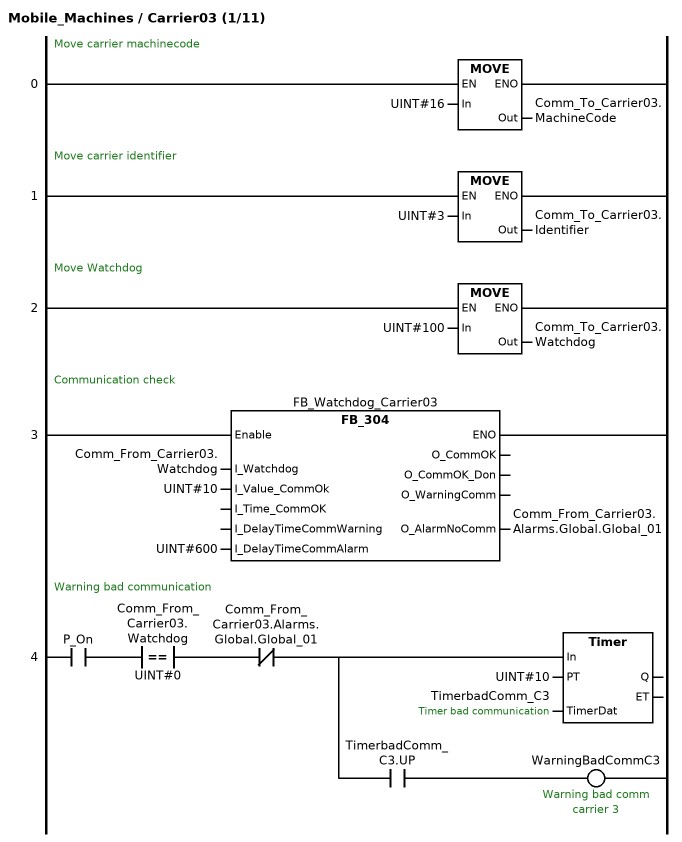
(* Rung 0: Move carrier machinecode *)
Comm_To_Carrier03.MachineCode := UINT#16;
(* Rung 1: Move carrier identifier *)
Comm_To_Carrier03.Identifier := UINT#3;
(* Rung 2: Move Watchdog *)
Comm_To_Carrier03.Watchdog := UINT#100;
(* Rung 3: Communication check *)
FB_Watchdog_Carrier03(Enable := TRUE, I_Watchdog := Comm_From_Carrier03.Watchdog, I_Value_CommOk := UINT#10, I_DelayTimeCommAlarm := UINT#600, O_AlarmNoComm => Comm_From_Carrier03.Alarms.Global.Global_01);
(* Rung 4: Warning bad communication *)
_p29 := P_On AND (Comm_From_Carrier03.Watchdog = UINT#0) AND NOT Comm_From_Carrier03.Alarms.Global.Global_01;
_t30 := Timer(In := _p29, PT := UINT#10, TimerDat := TimerbadComm_C3);
WarningBadCommC3 := _p29 AND TimerbadComm_C3.UP;

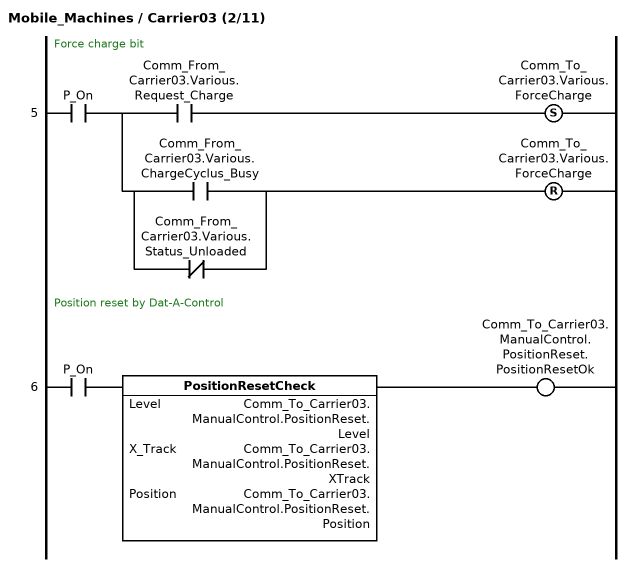
(* Rung 5: Force charge bit *)
IF P_On AND Comm_From_Carrier03.Various.Request_Charge THEN
    Comm_To_Carrier03.Various.ForceCharge := TRUE;
END_IF;
IF P_On AND (Comm_From_Carrier03.Various.ChargeCyclus_Busy OR NOT Comm_From_Carrier03.Various.Status_Unloaded) THEN
    Comm_To_Carrier03.Various.ForceCharge := FALSE;
END_IF;
(* Rung 6: Position reset by Dat-A-Control *)
Comm_To_Carrier03.ManualControl.PositionReset.PositionResetOk := P_On AND PositionResetCheck(Level := Comm_To_Carrier03.ManualControl.PositionReset.Level, X_Track := Comm_To_Carrier03.ManualControl.PositionReset.XTrack, Position := Comm_To_Carrier03.ManualControl.PositionReset.Position);

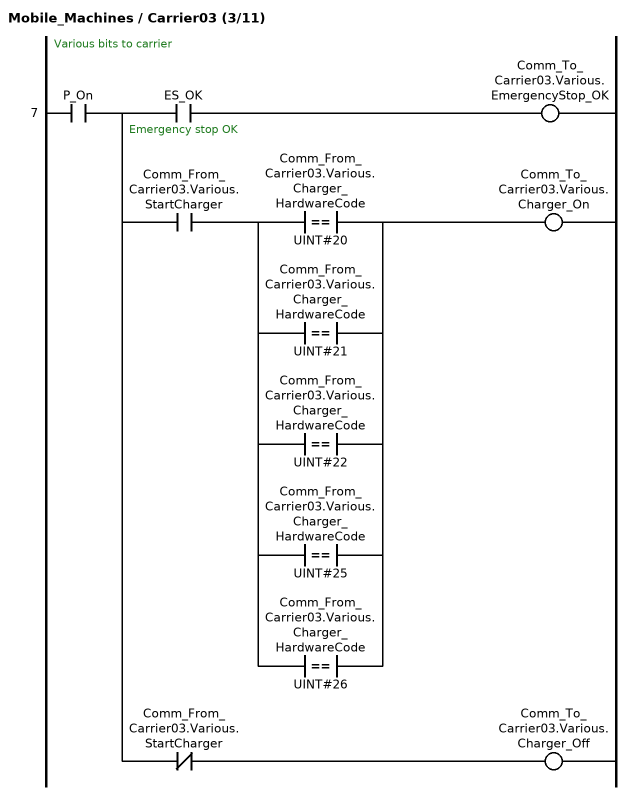
(* Rung 7: Various bits to carrier *)
Comm_To_Carrier03.Various.EmergencyStop_OK := P_On AND ES_OK;
Comm_To_Carrier03.Various.Charger_On := P_On AND Comm_From_Carrier03.Various.StartCharger AND ((Comm_From_Carrier03.Various.Charger_HardwareCode = UINT#20) OR (Comm_From_Carrier03.Various.Charger_HardwareCode = UINT#21) OR (Comm_From_Carrier03.Various.Charger_HardwareCode = UINT#22) OR (Comm_From_Carrier03.Various.Charger_HardwareCode = UINT#25) OR (Comm_From_Carrier03.Various.Charger_HardwareCode = UINT#26));
Comm_To_Carrier03.Various.Charger_Off := P_On AND NOT Comm_From_Carrier03.Various.StartCharger;

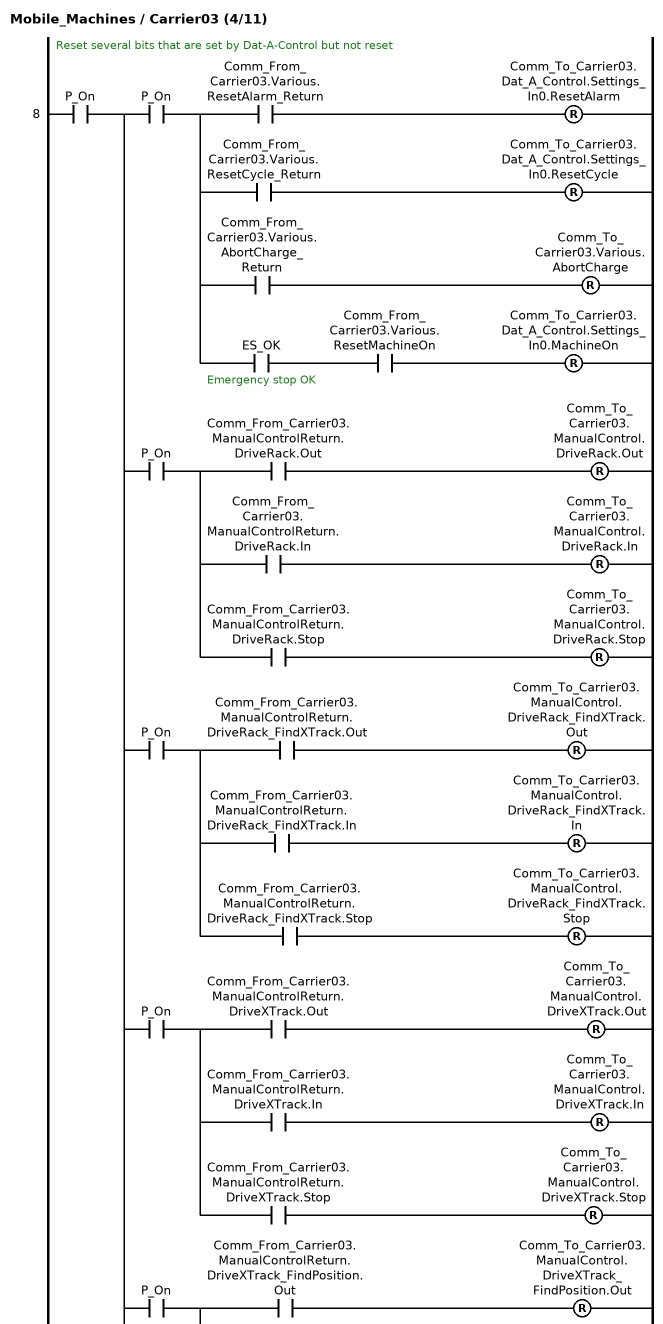

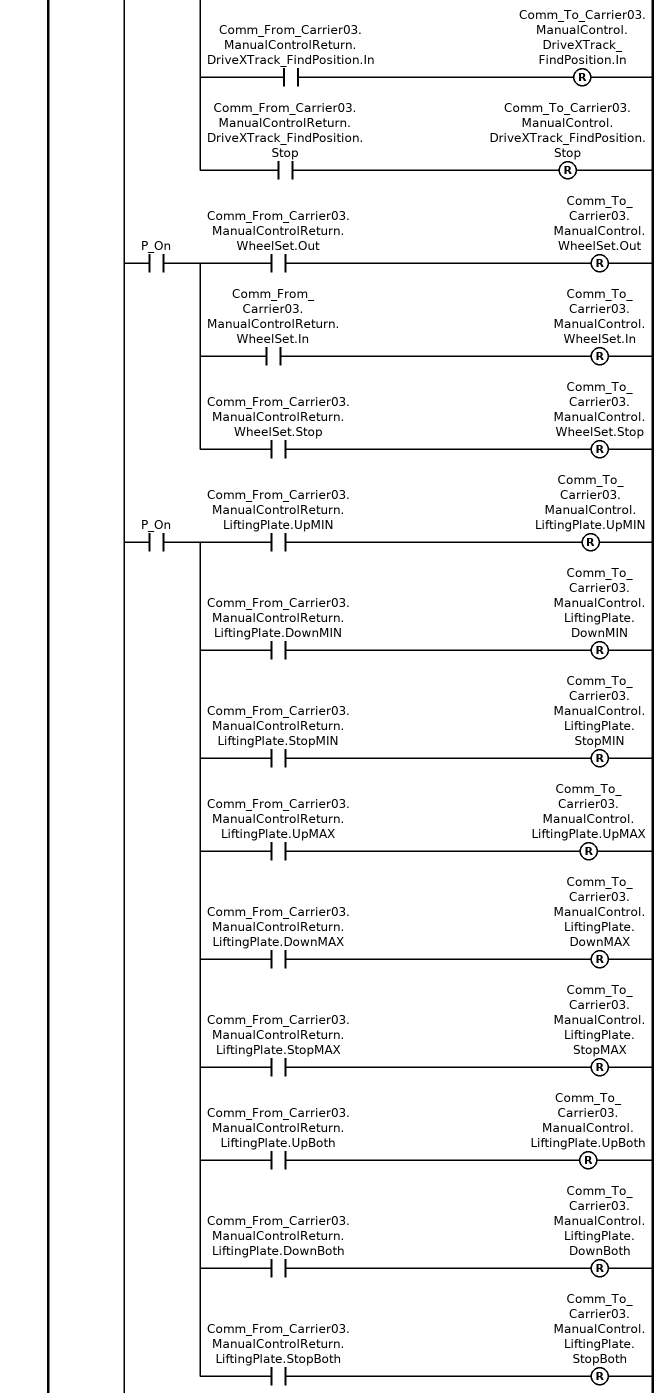

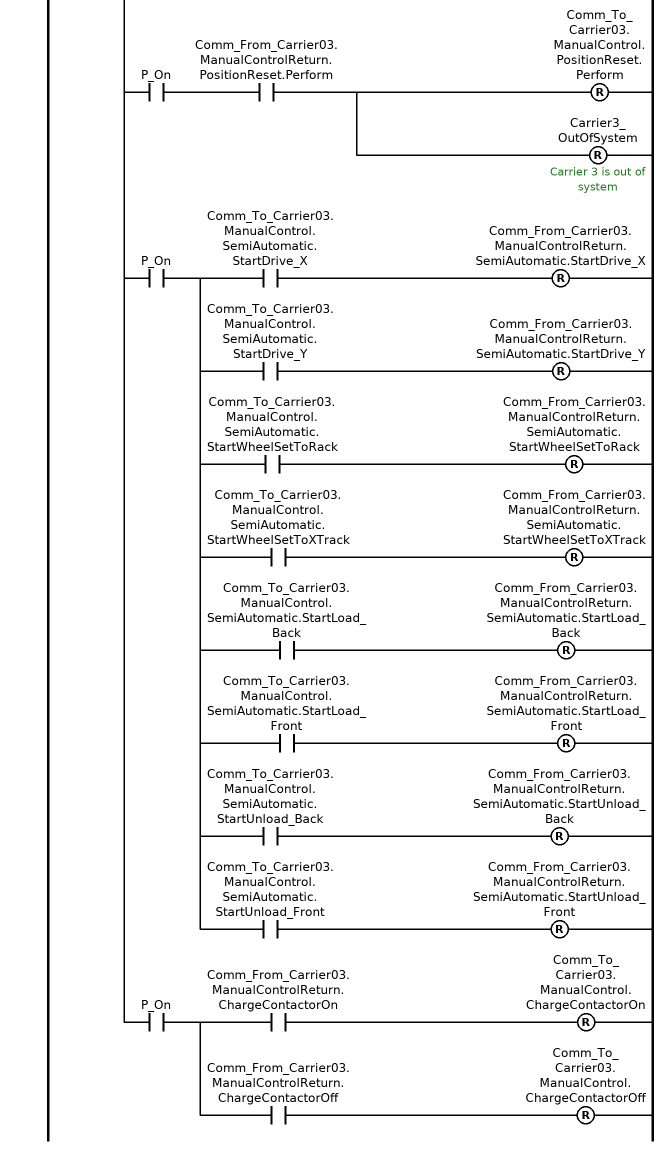
(* Rung 8: Reset several bits that are set by Dat-A-Control but not reset *)
IF P_On AND P_On AND Comm_From_Carrier03.Various.ResetAlarm_Return THEN
    Comm_To_Carrier03.Dat_A_Control.Settings_In0.ResetAlarm := FALSE;
END_IF;
IF P_On AND P_On AND Comm_From_Carrier03.Various.ResetCycle_Return THEN
    Comm_To_Carrier03.Dat_A_Control.Settings_In0.ResetCycle := FALSE;
END_IF;
IF P_On AND P_On AND Comm_From_Carrier03.Various.AbortCharge_Return THEN
    Comm_To_Carrier03.Various.AbortCharge := FALSE;
END_IF;
IF P_On AND P_On AND ES_OK AND Comm_From_Carrier03.Various.ResetMachineOn THEN
    Comm_To_Carrier03.Dat_A_Control.Settings_In0.MachineOn := FALSE;
END_IF;
IF P_On AND P_On AND Comm_From_Carrier03.ManualControlReturn.DriveRack.Out THEN
    Comm_To_Carrier03.ManualControl.DriveRack.Out := FALSE;
END_IF;
IF P_On AND P_On AND Comm_From_Carrier03.ManualControlReturn.DriveRack.In THEN
    Comm_To_Carrier03.ManualControl.DriveRack.In := FALSE;
END_IF;
IF P_On AND P_On AND Comm_From_Carrier03.ManualControlReturn.DriveRack.Stop THEN
    Comm_To_Carrier03.ManualControl.DriveRack.Stop := FALSE;
END_IF;
IF P_On AND P_On AND Comm_From_Carrier03.ManualControlReturn.DriveRack_FindXTrack.Out THEN
    Comm_To_Carrier03.ManualControl.DriveRack_FindXTrack.Out := FALSE;
END_IF;
IF P_On AND P_On AND Comm_From_Carrier03.ManualControlReturn.DriveRack_FindXTrack.In THEN
    Comm_To_Carrier03.ManualControl.DriveRack_FindXTrack.In := FALSE;
END_IF;
IF P_On AND P_On AND Comm_From_Carrier03.ManualControlReturn.DriveRack_FindXTrack.Stop THEN
    Comm_To_Carrier03.ManualControl.DriveRack_FindXTrack.Stop := FALSE;
END_IF;
IF P_On AND P_On AND Comm_From_Carrier03.ManualControlReturn.DriveXTrack.Out THEN
    Comm_To_Carrier03.ManualControl.DriveXTrack.Out := FALSE;
END_IF;
IF P_On AND P_On AND Comm_From_Carrier03.ManualControlReturn.DriveXTrack.In THEN
    Comm_To_Carrier03.ManualControl.DriveXTrack.In := FALSE;
END_IF;
IF P_On AND P_On AND Comm_From_Carrier03.ManualControlReturn.DriveXTrack.Stop THEN
    Comm_To_Carrier03.ManualControl.DriveXTrack.Stop := FALSE;
END_IF;
IF P_On AND P_On AND Comm_From_Carrier03.ManualControlReturn.DriveXTrack_FindPosition.Out THEN
    Comm_To_Carrier03.ManualControl.DriveXTrack_FindPosition.Out := FALSE;
END_IF;
IF P_On AND P_On AND Comm_From_Carrier03.ManualControlReturn.DriveXTrack_FindPosition.In THEN
    Comm_To_Carrier03.ManualControl.DriveXTrack_FindPosition.In := FALSE;
END_IF;
IF P_On AND P_On AND Comm_From_Carrier03.ManualControlReturn.DriveXTrack_FindPosition.Stop THEN
    Comm_To_Carrier03.ManualControl.DriveXTrack_FindPosition.Stop := FALSE;
END_IF;
IF P_On AND P_On AND Comm_From_Carrier03.ManualControlReturn.WheelSet.Out THEN
    Comm_To_Carrier03.ManualControl.WheelSet.Out := FALSE;
END_IF;
IF P_On AND P_On AND Comm_From_Carrier03.ManualControlReturn.WheelSet.In THEN
    Comm_To_Carrier03.ManualControl.WheelSet.In := FALSE;
END_IF;
IF P_On AND P_On AND Comm_From_Carrier03.ManualControlReturn.WheelSet.Stop THEN
    Comm_To_Carrier03.ManualControl.WheelSet.Stop := FALSE;
END_IF;
IF P_On AND P_On AND Comm_From_Carrier03.ManualControlReturn.LiftingPlate.UpMIN THEN
    Comm_To_Carrier03.ManualControl.LiftingPlate.UpMIN := FALSE;
END_IF;
IF P_On AND P_On AND Comm_From_Carrier03.ManualControlReturn.LiftingPlate.DownMIN THEN
    Comm_To_Carrier03.ManualControl.LiftingPlate.DownMIN := FALSE;
END_IF;
IF P_On AND P_On AND Comm_From_Carrier03.ManualControlReturn.LiftingPlate.StopMIN THEN
    Comm_To_Carrier03.ManualControl.LiftingPlate.StopMIN := FALSE;
END_IF;
IF P_On AND P_On AND Comm_From_Carrier03.ManualControlReturn.LiftingPlate.UpMAX THEN
    Comm_To_Carrier03.ManualControl.LiftingPlate.UpMAX := FALSE;
END_IF;
IF P_On AND P_On AND Comm_From_Carrier03.ManualControlReturn.LiftingPlate.DownMAX THEN
    Comm_To_Carrier03.ManualControl.LiftingPlate.DownMAX := FALSE;
END_IF;
IF P_On AND P_On AND Comm_From_Carrier03.ManualControlReturn.LiftingPlate.StopMAX THEN
    Comm_To_Carrier03.ManualControl.LiftingPlate.StopMAX := FALSE;
END_IF;
IF P_On AND P_On AND Comm_From_Carrier03.ManualControlReturn.LiftingPlate.UpBoth THEN
    Comm_To_Carrier03.ManualControl.LiftingPlate.UpBoth := FALSE;
END_IF;
IF P_On AND P_On AND Comm_From_Carrier03.ManualControlReturn.LiftingPlate.DownBoth THEN
    Comm_To_Carrier03.ManualControl.LiftingPlate.DownBoth := FALSE;
END_IF;
IF P_On AND P_On AND Comm_From_Carrier03.ManualControlReturn.LiftingPlate.StopBoth THEN
    Comm_To_Carrier03.ManualControl.LiftingPlate.StopBoth := FALSE;
END_IF;
_p31 := P_On AND P_On AND Comm_From_Carrier03.ManualControlReturn.PositionReset.Perform;
IF _p31 THEN
    Comm_To_Carrier03.ManualControl.PositionReset.Perform := FALSE;
    Carrier3_OutOfSystem := FALSE;
END_IF;
IF P_On AND P_On AND Comm_To_Carrier03.ManualControl.SemiAutomatic.StartDrive_X THEN
    Comm_From_Carrier03.ManualControlReturn.SemiAutomatic.StartDrive_X := FALSE;
END_IF;
IF P_On AND P_On AND Comm_To_Carrier03.ManualControl.SemiAutomatic.StartDrive_Y THEN
    Comm_From_Carrier03.ManualControlReturn.SemiAutomatic.StartDrive_Y := FALSE;
END_IF;
IF P_On AND P_On AND Comm_To_Carrier03.ManualControl.SemiAutomatic.StartWheelSetToRack THEN
    Comm_From_Carrier03.ManualControlReturn.SemiAutomatic.StartWheelSetToRack := FALSE;
END_IF;
IF P_On AND P_On AND Comm_To_Carrier03.ManualControl.SemiAutomatic.StartWheelSetToXTrack THEN
    Comm_From_Carrier03.ManualControlReturn.SemiAutomatic.StartWheelSetToXTrack := FALSE;
END_IF;
IF P_On AND P_On AND Comm_To_Carrier03.ManualControl.SemiAutomatic.StartLoad_Back THEN
    Comm_From_Carrier03.ManualControlReturn.SemiAutomatic.StartLoad_Back := FALSE;
END_IF;
IF P_On AND P_On AND Comm_To_Carrier03.ManualControl.SemiAutomatic.StartLoad_Front THEN
    Comm_From_Carrier03.ManualControlReturn.SemiAutomatic.StartLoad_Front := FALSE;
END_IF;
IF P_On AND P_On AND Comm_To_Carrier03.ManualControl.SemiAutomatic.StartUnload_Back THEN
    Comm_From_Carrier03.ManualControlReturn.SemiAutomatic.StartUnload_Back := FALSE;
END_IF;
IF P_On AND P_On AND Comm_To_Carrier03.ManualControl.SemiAutomatic.StartUnload_Front THEN
    Comm_From_Carrier03.ManualControlReturn.SemiAutomatic.StartUnload_Front := FALSE;
END_IF;
IF P_On AND P_On AND Comm_From_Carrier03.ManualControlReturn.ChargeContactorOn THEN
    Comm_To_Carrier03.ManualControl.ChargeContactorOn := FALSE;
END_IF;
IF P_On AND P_On AND Comm_From_Carrier03.ManualControlReturn.ChargeContactorOff THEN
    Comm_To_Carrier03.ManualControl.ChargeContactorOff := FALSE;
END_IF;

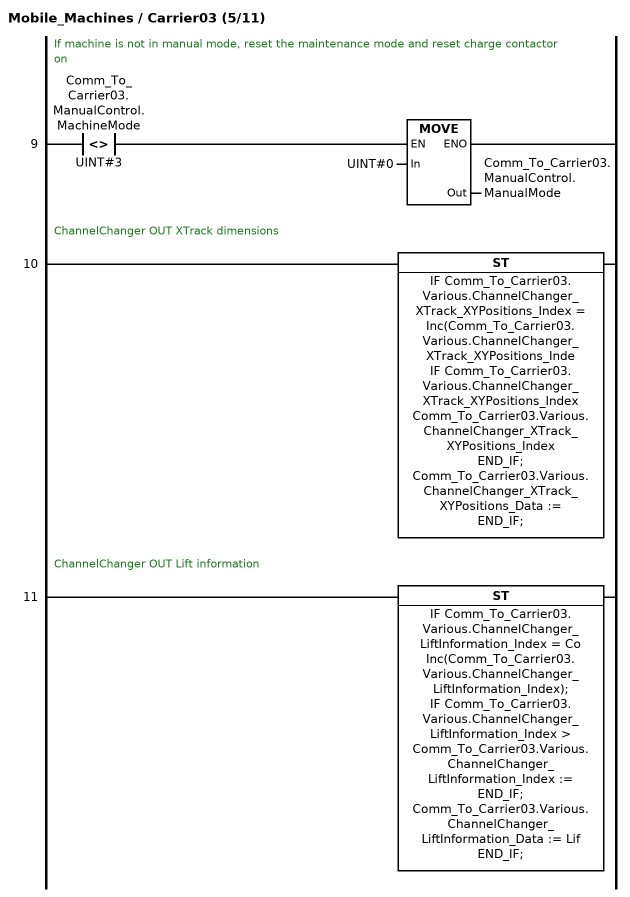
(* Rung 9: If machine is not in manual mode, reset the maintenance mode and reset charge contactor on *)
IF Comm_To_Carrier03.ManualControl.MachineMode <> UINT#3 THEN
    Comm_To_Carrier03.ManualControl.ManualMode := UINT#0;
END_IF;
(* Rung 10: ChannelChanger OUT XTrack dimensions *)
IF Comm_To_Carrier03.Various.ChannelChanger_XTrack_XYPositions_Index = Comm_From_Carrier03.Various.ChannelChanger_XTrack_XYPositions_Index THEN
	Inc(Comm_To_Carrier03.Various.ChannelChanger_XTrack_XYPositions_Index);
	IF Comm_To_Carrier03.Various.ChannelChanger_XTrack_XYPositions_Index > 199 THEN
		Comm_To_Carrier03.Various.ChannelChanger_XTrack_XYPositions_Index := 0;
	END_IF;
	Comm_To_Carrier03.Various.ChannelChanger_XTrack_XYPositions_Data := XTrack_XYPositions_Array[Comm_To_Carrier03.Various.ChannelChanger_XTrack_XYPositions_Index];
END_IF;
(* Rung 11: ChannelChanger OUT Lift information *)
IF Comm_To_Carrier03.Various.ChannelChanger_LiftInformation_Index = Comm_From_Carrier03.Various.ChannelChanger_LiftInformation_Index THEN
	Inc(Comm_To_Carrier03.Various.ChannelChanger_LiftInformation_Index);
	IF Comm_To_Carrier03.Various.ChannelChanger_LiftInformation_Index > 99 THEN
		Comm_To_Carrier03.Various.ChannelChanger_LiftInformation_Index := 0;
	END_IF;
	Comm_To_Carrier03.Various.ChannelChanger_LiftInformation_Data := Lift_Array[Comm_To_Carrier03.Various.ChannelChanger_LiftInformation_Index];
END_IF;

